// TIA Portal V20 export
VAR_GLOBAL   // PLC tag table "Part_Type"
END_VAR
VAR_GLOBAL CONSTANT   // user constants
   Part : Int := 1;
   ViceWithoutPart : Int := 2;
   Pallet : Int := 3;
   Gripper : Int := 4;
   ViceWithPart : Int := 5;
   TRAY : Int := 6;
END_VAR
